{attribute 'c++_compatible'}
FUNCTION_BLOCK UdpReceiver IMPLEMENTS ITcIoUdpProtocolRecv
VAR_INPUT
END_VAR
VAR_OUTPUT
END_VAR
VAR
	{attribute 'TcInitSymbol'}
	oid: OTCID; 
	ipUdp: 		ITcIoUdpProtocol;
	nUdpPort: 	UINT := 10000;
	nReceivedPakets: UINT;
	lastReceivedIP : IpAdrUnion; 
	hrInit : HRESULT;

END_VAR

METHOD CyclicUpdate : BOOL
VAR_INPUT
END_VAR
IF ipUdp <> 0 THEN
	ipUdp.CheckReceived();
END_IF
END_METHOD

METHOD FB_exit : BOOL
VAR_INPUT
	bInCopyCode : BOOL; // if TRUE, the exit method is called for exiting an instance that is copied afterwards (online change).
END_VAR
IF (NOT bInCopyCode AND ipUdp <> 0) THEN //Shutdown
	ipUdp.UnregisterReceiver(nUdpPort);
	FW_SafeRelease(ADR(ipUdp));
	FB_exit := TRUE;
ELSE
	FB_exit := FALSE;
END_IF
END_METHOD

METHOD FB_init : BOOL
VAR_INPUT
	bInitRetains : BOOL; // if TRUE, the retain variables are initialized (warm start / cold start)
	bInCopyCode : BOOL;  // if TRUE, the instance afterwards gets moved into the copy code (online change)
END_VAR
VAR
	//ipSrv: ITComObjectServer;
END_VAR
IF NOT bInCopyCode THEN // no online change
	IF ipUdp = 0 AND oid <> 0 THEN
	 hrInit := FW_ObjMgr_GetObjectInstance(oid:=oid, iid:=TC_GLOBAL_IID_LIST.IID_ITcIoUdpProtocol, pipUnk:=ADR(ipUdp) );
		IF SUCCEEDED(hrInit) THEN 
			IF SUCCEEDED(ipUdp.RegisterReceiver(nUdpPort, THIS^)) THEN //open port
				FB_init := TRUE;
			ELSE 
				FB_init := FALSE; 
				FW_SafeRelease(ADR(ipUdp));
			END_IF
		END_IF
	ELSIF oid = 0 THEN 
		FB_init := FALSE; 
		hrInit := ERR_INVALID_PARAM; 				
	END_IF
END_IF
END_METHOD

METHOD FB_reinit : BOOL
VAR_INPUT
END_VAR
IF (ipUdp <> 0) THEN 
  ipUdp.RegisterReceiver(nUdpPort, THIS^);
  FB_reinit := TRUE; 
END_IF
END_METHOD

{attribute 'object_name' := 'ReceiveData'}
{attribute 'c++_compatible'}
{attribute 'pack_mode' := '4'}
{attribute 'show'}
{attribute 'minimal_input_size' := '4'}
METHOD ReceiveData : HRESULT
VAR_INPUT
	ipAddr	: UDINT;
	udpDestPort	: UINT;
	udpSrcPort	: UINT;
	nData	: UDINT;
	pData	: PVOID;
	pVlan	: POINTER TO ETYPE_VLAN_HEADER := 0;
END_VAR
nReceivedPakets := nReceivedPakets+1;
lastReceivedIP.ipadrIPStack := ipAddr;
IF ipUdp <> 0 THEN
	ipUdp.SendData(ipAddr, udpSrcPort, udpDestPort, nData, pData, TRUE, 0); // send data back
END_IF
END_METHOD

{attribute 'object_name' := 'TcAddRef'}
{attribute 'c++_compatible'}
{attribute 'pack_mode' := '4'}
{attribute 'show'}
{attribute 'minimal_input_size' := '4'}
METHOD TcAddRef : UDINT
END_METHOD

{attribute 'object_name' := 'TcQueryInterface'}
{attribute 'c++_compatible'}
{attribute 'pack_mode' := '4'}
{attribute 'show'}
{attribute 'minimal_input_size' := '4'}
METHOD TcQueryInterface : HRESULT
VAR_INPUT
	iid	: REFERENCE TO IID;
	pipItf	: POINTER TO PVOID;
END_VAR
VAR
   ipUdpRecv : ITcIoUdpProtocolRecv;
   ipUnknown : ITcUnknown;   
END_VAR
IF GuidsEqual(ADR(iid), ADR(TC_GLOBAL_IID_LIST.IID_ITcIoUdpProtocolRecv)) THEN
   ipUdpRecv := THIS^; // cast to interface pointer
   pipItf^ := ITCUNKNOWN_TO_PVOID(ipUdpRecv);
   TcAddRef();
   TcQueryInterface := S_OK;
ELSIF GuidsEqual(ADR(iid), ADR(TC_GLOBAL_IID_LIST.IID_ITcUnknown)) THEN
   ipUnknown := THIS^; // cast to interface pointer
   pipItf^ := ITCUNKNOWN_TO_PVOID(ipUnknown);
   TcAddRef();
   TcQueryInterface := S_OK;
ELSE
   TcQueryInterface := E_HRESULTAdsErr.NOINTERFACE ; //Call super if this fb extends some other
END_IF
END_METHOD

{attribute 'object_name' := 'TcRelease'}
{attribute 'c++_compatible'}
{attribute 'pack_mode' := '4'}
{attribute 'show'}
{attribute 'minimal_input_size' := '4'}
METHOD TcRelease : UDINT
END_METHOD

END_FUNCTION_BLOCK

(* stored: Version 1.1.0.1
   POU UdpReceiver: Id {3b4b2ae9-c069-42e3-9b69-f42439287066}, SpecialFunc None
   Method CyclicUpdate: Id {169c50b7-1a40-4541-9526-3b8a41abf2d1}
   Method FB_exit: Id {0258286a-12f2-440d-8e54-fd50a76e4c92}
   Method FB_init: Id {3f9ab792-5971-4b0c-a6bc-dc33a9b3d66e}
   Method FB_reinit: Id {230ea14e-9797-48ee-9586-6313ceab7837}
   Method ReceiveData: Id {cb5b89bf-a2d8-4ac3-bd40-64d876626d0f}
   Method TcAddRef: Id {2d410f6b-c6bd-4033-8c18-8496c8308aff}
   Method TcQueryInterface: Id {0544c61f-9985-4e5f-b52a-347332675914}
   Method TcRelease: Id {bb0886f8-6f09-4d5a-835f-a451f23c160e} *)
